(* IEC 61131-3 sources: eCockpitGit/test_project/src/%F%00 Library/%F%Common Functions/%F%Bits/%F%Bit Set Part In Place, 8 files *)

(* ---- %POU%FU_bBitPart.st ---- *)
//This function changed only the needed bits of a variable
// |**Version**|**Author**| **Date** |**Changes**
// | 1         | NSN      | 16-03-22 | Creation
FUNCTION FU_bBitPart : BOOL
VAR_IN_OUT
	valueChange		:BYTE;		//Variable to change
END_VAR
VAR_INPUT
	value			:BYTE;		//Value to change bits to
	amount			:BYTE;		//Amount of bits to change
	offset			:BYTE;		//Offset in variable to change bits at
END_VAR
(*%!%__DELIMITER__%!%*)
valueChange		:=		(valueChange AND ROL(GConstants.binaryInvMaskByte[amount],offset)) OR SHL(value AND GConstants.binaryMaskByte[amount],offset);

(* ---- %POU%FU_diBitPart.st ---- *)
//This function changed only the needed bits of a variable
// |**Version**|**Author**| **Date** |**Changes**
// | 1         | NSN      | 16-03-22 | Creation
FUNCTION FU_diBitPart : BOOL
VAR_IN_OUT
	valueChange		:DINT;		//Variable to change
END_VAR
VAR_INPUT
	value			:DINT;		//Value to change bits to
	amount			:BYTE;		//Amount of bits to change
	offset			:BYTE;		//Offset in variable to change bits at
END_VAR
(*%!%__DELIMITER__%!%*)
valueChange		:=		TO_DINT((TO_UDINT(valueChange) AND ROL(TO_UDINT(GConstants.binaryInvMaskDint[amount]),offset)) OR SHL(TO_UDINT(value) AND TO_UDINT(GConstants.binaryMaskDint[amount]),offset));

(* ---- %POU%FU_dwBitPart.st ---- *)
//This function changed only the needed bits of a variable
// |**Version**|**Author**| **Date** |**Changes**
// | 1         | NSN      | 16-03-22 | Creation
FUNCTION FU_dwBitPart : BOOL
VAR_IN_OUT
	valueChange		:DWORD;		//Variable to change
END_VAR
VAR_INPUT
	value			:DWORD;		//Value to change bits to
	amount			:BYTE;		//Amount of bits to change
	offset			:BYTE;		//Offset in variable to change bits at
END_VAR
(*%!%__DELIMITER__%!%*)
valueChange		:=		(valueChange AND ROL(GConstants.binaryInvMaskDWord[amount],offset)) OR SHL(value AND GConstants.binaryMaskDWord[amount],offset);

(* ---- %POU%FU_iBitPart.st ---- *)
//This function changed only the needed bits of a variable
// |**Version**|**Author**| **Date** |**Changes**
// | 1         | NSN      | 16-03-22 | Creation
FUNCTION FU_iBitPart : BOOL
VAR_IN_OUT
	valueChange		:INT;		//Variable to change
END_VAR
VAR_INPUT
	value			:INT;		//Value to change bits to
	amount			:BYTE;		//Amount of bits to change
	offset			:BYTE;		//Offset in variable to change bits at
END_VAR
(*%!%__DELIMITER__%!%*)
valueChange		:=		TO_INT((TO_UINT(valueChange) AND ROL(TO_UINT(GConstants.binaryInvMaskInt[amount]),offset)) OR SHL(TO_UINT(value) AND TO_UINT(GConstants.binaryMaskInt[amount]),offset));

(* ---- %POU%FU_liBitPart.st ---- *)
//This function changed only the needed bits of a variable
// |**Version**|**Author**| **Date** |**Changes**
// | 1         | NSN      | 16-03-22 | Creation
FUNCTION FU_liBitPart : BOOL
VAR_IN_OUT
	valueChange		:LINT;		//Variable to change
END_VAR
VAR_INPUT
	value			:LINT;		//Value to change bits to
	amount			:BYTE;		//Amount of bits to change
	offset			:BYTE;		//Offset in variable to change bits at
END_VAR
(*%!%__DELIMITER__%!%*)
valueChange		:=		TO_LINT((TO_ULINT(valueChange) AND ROL(TO_ULINT(GConstants.binaryInvMaskLint[amount]),offset)) OR SHL(TO_ULINT(value) AND TO_ULINT(GConstants.binaryMaskLint[amount]),offset));

(* ---- %POU%FU_lwBitPart.st ---- *)
//This function changed only the needed bits of a variable
// |**Version**|**Author**| **Date** |**Changes**
// | 1         | NSN      | 16-03-22 | Creation
FUNCTION FU_lwBitPart : BOOL
VAR_IN_OUT
	valueChange		:LWORD;		//Variable to change
END_VAR
VAR_INPUT
	value			:LWORD;		//Value to change bits to
	amount			:BYTE;		//Amount of bits to change
	offset			:BYTE;		//Offset in variable to change bits at
END_VAR
(*%!%__DELIMITER__%!%*)
valueChange		:=		(valueChange AND ROL(GConstants.binaryInvMaskLWord[amount],offset)) OR SHL(value AND GConstants.binaryMaskLWord[amount],offset);

(* ---- %POU%FU_siBitPart.st ---- *)
//This function changed only the needed bits of a variable
// |**Version**|**Author**| **Date** |**Changes**
// | 1         | NSN      | 16-03-22 | Creation
FUNCTION FU_siBitPart : BOOL
VAR_IN_OUT
	valueChange		:SINT;		//Variable to change
END_VAR
VAR_INPUT
	value			:SINT;		//Value to change bits to
	amount			:BYTE;		//Amount of bits to change
	offset			:BYTE;		//Offset in variable to change bits at
END_VAR
(*%!%__DELIMITER__%!%*)
valueChange		:=		TO_SINT((TO_USINT(valueChange) AND ROL(TO_USINT(GConstants.binaryInvMaskSint[amount]),offset)) OR SHL(TO_USINT(value) AND TO_USINT(GConstants.binaryMaskSint[amount]),offset));

(* ---- %POU%FU_wBitPart.st ---- *)
//This function changed only the needed bits of a variable
// |**Version**|**Author**| **Date** |**Changes**
// | 1         | NSN      | 16-03-22 | Creation
FUNCTION FU_wBitPart : BOOL
VAR_IN_OUT
	valueChange		:WORD;		//Variable to change
END_VAR
VAR_INPUT
	value			:WORD;		//Value to change bits to
	amount			:BYTE;		//Amount of bits to change
	offset			:BYTE;		//Offset in variable to change bits at
END_VAR
(*%!%__DELIMITER__%!%*)
valueChange		:=		(valueChange AND ROL(GConstants.binaryInvMaskWord[amount],offset)) OR SHL(value AND GConstants.binaryMaskWord[amount],offset);
